// TIA Portal V19 export
VAR_GLOBAL   // PLC tag table "A03_304"
   A0303_Navetta_Ax_Scarico_Testa_Ls_Minimo AT %I358.7 : Bool;   // 2432SQ1
   A0303_Navetta_Ax_Scarico_Testa_Ls_Massimo AT %I359.0 : Bool;   // 2432SQ2
   A0303_Navetta_Paletto_Interno_Testa_Ls_Rest AT %I359.1 : Bool;   // 2440SQ1
   A0303_Navetta_Paletto_Interno_Testa_Ls_Work AT %I359.2 : Bool;   // 2440SQ2
   A0303_Navetta_Paletto_Interno_Testa_V_Rest AT %Q364.0 : Bool;   // 2440YV1
   A0303_Navetta_Paletto_Interno_Testa_V_Work AT %Q364.1 : Bool;   // 2440YV2
   A0303_Navetta_Paletto_Interno_Testa_SbloccaggioStelo_V_Work AT %Q364.2 : Bool;   // 2440YV3 (0 = BLOCCATO ; 1 = SBLOCCATO)
   A0303_Navetta_Paletto_Esterno_Testa_Ls_Rest AT %I359.3 : Bool;   // 2442SQ1
   A0303_Navetta_Paletto_Esterno_Testa_Ls_Work AT %I359.4 : Bool;   // 2442SQ2
   A0303_Navetta_Paletto_Esterno_Testa_V_Rest AT %Q364.3 : Bool;   // 2442YV1
   A0303_Navetta_Paletto_Esterno_Testa_V_Work AT %Q364.4 : Bool;   // 2442YV2
   A0303_Navetta_Paletto_Esterno_Testa_SbloccaggioStelo_V_Work AT %Q364.5 : Bool;   // 2442YV3 (0 = BLOCCATO ; 1 = SBLOCCATO)
   A0303_Navetta_Ax_Scarico_Coda_Ls_Minimo AT %I308.7 : Bool;   // 2462SQ1
   A0303_Navetta_Ax_Scarico_Coda_Ls_Massimo AT %I309.0 : Bool;   // 2462SQ2
   A0303_Navetta_Paletto_Interno_Coda_Ls_Rest AT %I309.1 : Bool;   // 2470SQ1
   A0303_Navetta_Paletto_Interno_Coda_Ls_Work AT %I309.2 : Bool;   // 2470SQ2
   A0303_Navetta_Paletto_Interno_Coda_V_Rest AT %Q313.4 : Bool;   // 2470YV1
   A0303_Navetta_Paletto_Interno_Coda_V_Work AT %Q313.5 : Bool;   // 2470YV2
   A0303_Navetta_Paletto_Interno_Coda_SbloccaggioStelo_V_Work AT %Q313.6 : Bool;   // 2470YV3 (0 = BLOCCATO ; 1 = SBLOCCATO)
   A0303_Navetta_Paletto_Esterno_Coda_Ls_Rest AT %I309.3 : Bool;   // 2472SQ1
   A0303_Navetta_Paletto_Esterno_Coda_Ls_Work AT %I309.4 : Bool;   // 2472SQ2
   A0303_Navetta_Paletto_Esterno_Coda_V_Rest AT %Q313.7 : Bool;   // 2472YV1
   A0303_Navetta_Paletto_Esterno_Coda_V_Work AT %Q314.0 : Bool;   // 2472YV2
   A0303_Navetta_Paletto_Esterno_Coda_SbloccaggioStelo_V_Work AT %Q314.1 : Bool;   // 2472YV3 (0 = BLOCCATO ; 1 = SBLOCCATO)
   A0303_Phc_1_Controllo_Pacco_In_Carico AT %I359.5 : Bool;   // 2490BF1
   A0303_Phc_2_Controllo_Pacco_In_Carico AT %I359.6 : Bool;   // 2490BF2
   A0303_Phc_1_Controllo_Pacco_In_Scarico AT %I359.7 : Bool;   // 2500BF1
   A0303_Phc_2_Controllo_Pacco_In_Scarico AT %I360.0 : Bool;   // 2500BF2
   A0302_Centratori_Centraggio_2_Centrale_V_Basso AT %Q314.2 : Bool;   // 2022YV1
   A0302_Centratori_Centraggio_2_Centrale_V_Alto AT %Q314.3 : Bool;   // 2022YV2
   A0302_Centratori_Centraggio_2_Centrale_V_Aperto AT %Q314.4 : Bool;   // 2022YV3
   A0302_Centratori_Centraggio_2_Centrale_V_Chiuso AT %Q314.5 : Bool;   // 2022YV4
   A0302_Centratori_Centraggio_3_Testa_V_Basso AT %Q314.6 : Bool;   // 2024YV1
   A0302_Centratori_Centraggio_3_Testa_V_Alto AT %Q314.7 : Bool;   // 2024YV2
   A0302_Centratori_Centraggio_3_Testa_V_Aperto AT %Q315.0 : Bool;   // 2024YV3
   A0302_Centratori_Centraggio_3_Testa_V_Chiuso AT %Q315.1 : Bool;   // 2024YV4
END_VAR
